FUNCTION_BLOCK Person_Object EXTENDS TcoCore.TcoObject

METHOD Accept : BOOL
VAR_INPUT
END_VAR
END_METHOD

METHOD Refuse : BOOL
VAR_INPUT
END_VAR
END_METHOD

METHOD PUBLIC RequestForFavor
VAR_INPUT
	inRequestedFavor	:	STRING;
	inReturnFavor		:	STRING;
END_VAR
END_METHOD

END_FUNCTION_BLOCK

(* stored: Version 1.1.0.1, ProductVersion 3.1.4024.6
   POU Person_Object: Id {7dea4e2d-f024-0ba8-2c2e-ea35736e744d}, SpecialFunc None
   Method Accept: Id {44c4e924-54f1-0a50-03f2-592c994e5489}
   Method Refuse: Id {3778f75f-808b-0091-0d24-ae374b268cd1}
   Method RequestForFavor: Id {cf31844f-f21f-05a5-08eb-2ab3e61668a0} *)
